FUNCTION_BLOCK FB_SaMElementAborting EXTENDS FB_SaMElement
VAR
END_VAR

METHOD FB_init : BOOL
VAR_INPUT
	bInitRetains : BOOL; // if TRUE, the retain variables are initialized (warm start / cold start)
	bInCopyCode : BOOL;  // if TRUE, the instance afterwards gets moved into the copy code (online change)
END_VAR
THIS^.bTypeActive		:= TRUE;

THIS^.SetText (eLocation := E_BaseLocation.pl, wsDescription := "Przerywanie");
THIS^.SetText (eLocation := E_BaseLocation.en, wsDescription := "Aborting");
THIS^.SetText (eLocation := E_BaseLocation.de, wsDescription := "Abbruch");
THIS^.SetName (stName := THIS^.GetTexts ());
END_METHOD

METHOD public GetNextState : E_BaseMachineState
VAR_INPUT
END_VAR
GetNextState		:= E_BaseMachineState.Aborted;
END_METHOD

METHOD PUBLIC InvokeStateForTopElement : BOOL
VAR_INPUT
	itfTopElement		: ITF_BaseSaMStateMethod;
END_VAR
InvokeStateForTopElement	:= itfTopElement.SP_Aborting ();
END_METHOD

END_FUNCTION_BLOCK

(* stored: Version 1.1.0.1
   POU FB_SaMElementAborting: Id {c7d1042c-68f1-06d1-0ebb-5647496def75}, SpecialFunc None
   Method FB_init: Id {3dcda7e9-5af7-02bf-2491-f86b8526366c}
   Method GetNextState: Id {f3463331-6ab7-02b0-3b74-740734d48987}
   Method InvokeStateForTopElement: Id {acd4c272-a1bc-0c6c-3afb-6c54425fb879} *)
